Staubli VAL3: setValue.pgx

public program setValue(num x_nValue, num x_nIndex, num x_nValue1)
begin
  // set the value
  // saveAxis[x_nIndex].nValue=x_nValue
  nSaveaxis[x_nIndex]=x_nValue
  nSaveaxis1[x_nIndex]=x_nValue1
end
